{attribute 'qualified_only'}
//{attribute 'strict'}
TYPE E_CAMERA_DeviceType :    (*tAcquisitionTime - to be secured*)
(
	NONE,
	MV420_F,			//F -> Full resolution
	MV420_H,			//H -> Half resolution
	MV440SR_F,
	MV440SR_H,
	MV440HR_F,
	MV440HR_H,
	MV440UR_F,
	MV440UR_H,
	MV540S_F,
	MV540S_H,
	MV540H_F,
	MV540H_H,
	MV560U_F,
	MV560U_H,
	V430F	(*Omron*)

);
END_TYPE

(* stored: Version 1.1.0.1
   DUT E_CAMERA_DeviceType: Id {7780f542-f378-428a-a43c-02ed1d3c764f} *)
